(* Logix 5000 project; controller FRCFMS vendor 1 type 14 code 150 rev 33.11; software revision 33.00; part 2 of 3 *)
(* tags used below, declared in another part *)
   Additional_len : INT;
   Additional_len_read : INT;
   buff_bit_index : DINT;
   buff_byte_index : DINT;
   CMD_END : DINT;
   CMD_IN : DINT;
   CMD_LEN : DINT;
   CMD_LEN2 : INT;
   CMD_START : DINT;
   Coil_Byte_Count : DINT;
   coil_wr_index : DINT;
   Data_Received : BOOL;
   Found : BOOL;
   INT_DATA_IN : INT;
   INT_IN : INT;
   INT_STR_OUT : STRING;
   Listen_Retry_Tmr : TIMER;
   Listen_Socket_Lost : BOOL;
   Log_Old : DINT;
   Main_Read_Buffer : STR_4096[20];
   mb_bit_index : DINT;
   MB_Resp_Data : STR_462;
   MB_TMP_INT : INT;
   Modbus_Bytes : DINT;
   Modbus_CMD_Len : INT;
   Modbus_Cmd_String : STR_462;
   Modbus_ID : STRING;
   Modbus_Packet : STR_462;
   Modbus_resp_Str : STR_462;
   Modbus_Ret_CMD : STRING;
   Modbus_Ret_len : STRING;
   Modbus_Start : INT;
   Modbus_Unit : STRING;
   Next_Write : BOOL[32];
   No_Open_Sockets : BOOL;
   Nothing : BOOL;
   ONS : BOOL[64];
   RetryCreateSock : TIMER;
   RG_4x_Pos : DINT;
   RW_Instance : INT[20];
   RW_Select : DINT;
   Startup_Timer : TIMER;
   Str_Out : STR_1;
   String_Pos : INT;
   testint : DINT;
   Valid : BOOL[32];
   Valid_CMD : BOOL[32];
   Valid_Command : BOOL;
   Valid_End : BOOL;
   Valid_Len : BOOL;
   Valid_Start_Addr : BOOL;
   Valid_Value_05 : BOOL;
   W_Log_Accept : ALIAS FOR MBTU_Log_Enable.2;
   W_Log_Attribute : ALIAS FOR MBTU_Log_Enable.6;
   W_Log_Create : ALIAS FOR MBTU_Log_Enable.0;
   W_Log_Delete : ALIAS FOR MBTU_Log_Enable.5;
   W_Log_Errors : ALIAS FOR MBTU_Log_Enable.7;
   W_Log_Open : ALIAS FOR MBTU_Log_Enable.1;
   W_Log_Read : ALIAS FOR MBTU_Log_Enable.3;
   W_Log_Write : ALIAS FOR MBTU_Log_Enable.4;
   MBTI_Change_Log_MSG : MESSAGE;
   MBTI_Conn_Acc_Timeout_MSG : MESSAGE;
   MBTI_Conn_Accept_MSG : MESSAGE;
   MBTI_ConnectionsLastErrors : DINT;
   MBTI_Create_Sock_MSG : MESSAGE;
   MBTI_Delete_All_MSG : MESSAGE;
   MBTI_Instance : DINT;
   MBTI_Read_Data_MSG_00 : MESSAGE;
   MBTI_Read_Data_MSG_01 : MESSAGE;
   MBTI_Read_Data_MSG_02 : MESSAGE;
   MBTI_Read_Data_MSG_03 : MESSAGE;
   MBTI_Read_Data_MSG_04 : MESSAGE;
   MBTI_Read_Data_MSG_05 : MESSAGE;
   MBTI_Read_Data_MSG_06 : MESSAGE;
   MBTI_Read_Data_MSG_07 : MESSAGE;
   MBTI_Read_Data_MSG_08 : MESSAGE;
   MBTI_Read_Data_MSG_09 : MESSAGE;
   MBTI_Read_Done : BOOL[32];
   MBTI_Read_Resp : READ_RESP_STR[10];
   MBTI_RW_Inactivity_MSG : MESSAGE;
   MBTI_Sock_Accept_Resp : AcceptResponse;
   MBTI_Total_Open : INT;
   MBTI_Total_Open_MSG : MESSAGE;
   MBTI_Write_Data_MSG_00 : MESSAGE;
   MBTI_Write_Data_MSG_01 : MESSAGE;
   MBTI_Write_Data_MSG_02 : MESSAGE;
   MBTI_Write_Data_MSG_03 : MESSAGE;
   MBTI_Write_Data_MSG_04 : MESSAGE;
   MBTI_Write_Data_MSG_05 : MESSAGE;
   MBTI_Write_Data_MSG_06 : MESSAGE;
   MBTI_Write_Data_MSG_07 : MESSAGE;
   MBTI_Write_Data_MSG_08 : MESSAGE;
   MBTI_Write_Data_MSG_09 : MESSAGE;
   MBTI_Write_Data_Out : WRT_DATA[10];
   MBTU_Enable_MBTCP : BOOL;
   MBTU_EnetModulePort : STRING;
   MBTU_Log_Enable : DINT;
   MBTU_MB_0xx : BOOL[256];
   MBTU_MB_4xx : INT[100];
(* ModbusSlaveTCP, continued *)

ROUTINE _SUB_4x_WR   (* ladder *)
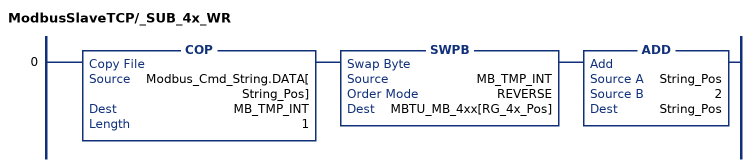
   0: COP(Modbus_Cmd_String.DATA[String_Pos],MB_TMP_INT,1)SWPB(MB_TMP_INT,REVERSE,MBTU_MB_4xx[RG_4x_Pos])ADD(String_Pos,2,String_Pos);
END_ROUTINE

ROUTINE _SUB_Byte2ST   (* ladder *)
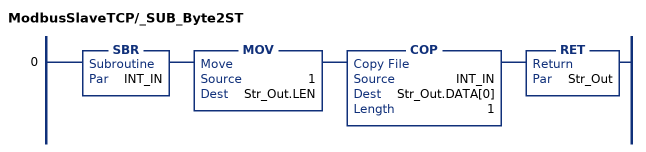
   0: SBR(INT_IN)MOV(1,Str_Out.LEN)COP(INT_IN,Str_Out.DATA[0],1)RET(Str_Out);
END_ROUTINE

ROUTINE _SUB_Int2ST   (* ladder *)
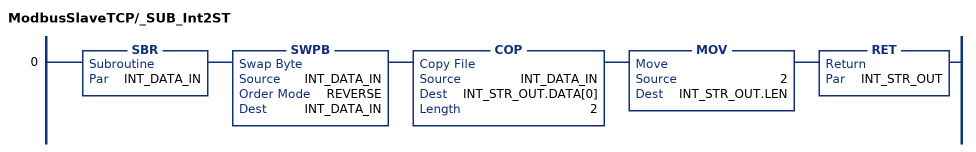
   0: SBR(INT_DATA_IN)SWPB(INT_DATA_IN,REVERSE,INT_DATA_IN)COP(INT_DATA_IN,INT_STR_OUT.DATA[0],2)MOV(2,INT_STR_OUT.LEN)RET(INT_STR_OUT);
END_ROUTINE

ROUTINE _SUB_SET_PATH   (* ladder *)
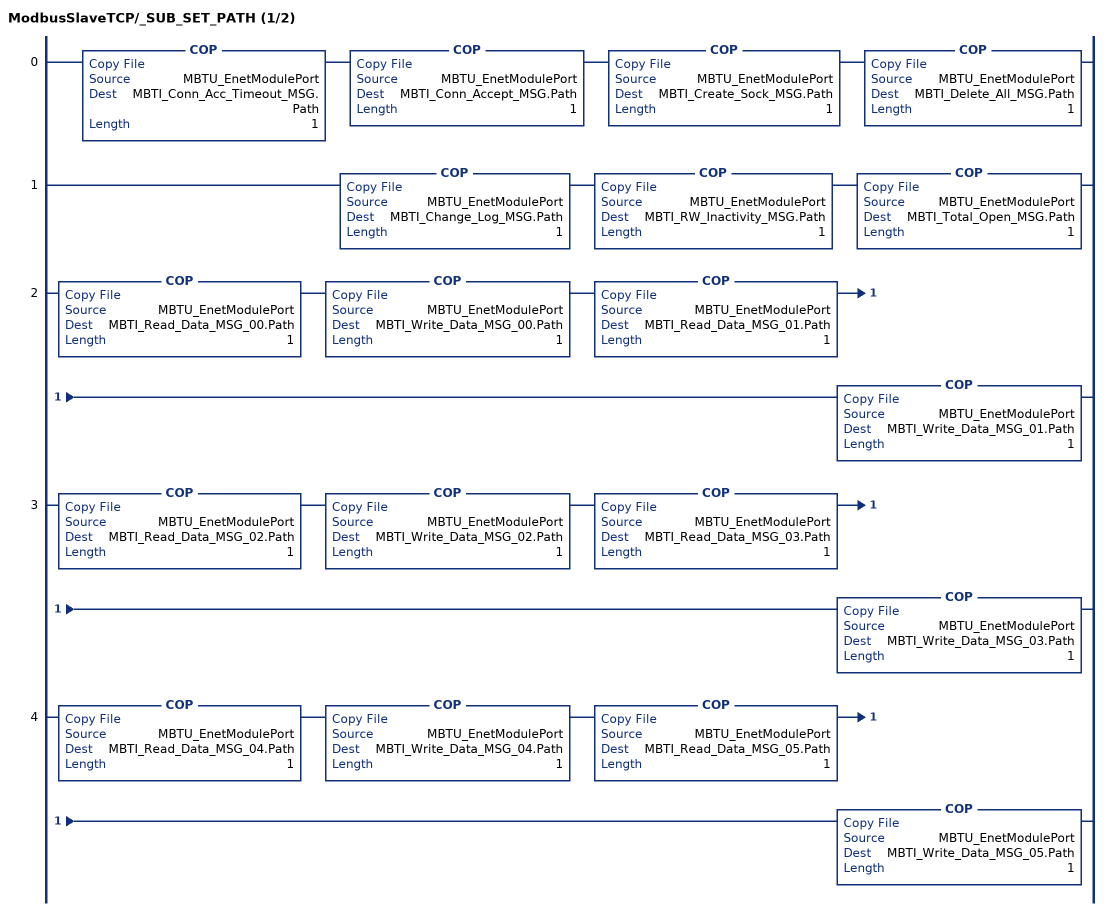
   0: COP(MBTU_EnetModulePort,MBTI_Conn_Acc_Timeout_MSG.Path,1)COP(MBTU_EnetModulePort,MBTI_Conn_Accept_MSG.Path,1)COP(MBTU_EnetModulePort,MBTI_Create_Sock_MSG.Path,1)COP(MBTU_EnetModulePort,MBTI_Delete_All_MSG.Path,1);
   1: COP(MBTU_EnetModulePort,MBTI_Change_Log_MSG.Path,1)COP(MBTU_EnetModulePort,MBTI_RW_Inactivity_MSG.Path,1)COP(MBTU_EnetModulePort,MBTI_Total_Open_MSG.Path,1);
   2: COP(MBTU_EnetModulePort,MBTI_Read_Data_MSG_00.Path,1)COP(MBTU_EnetModulePort,MBTI_Write_Data_MSG_00.Path,1)COP(MBTU_EnetModulePort,MBTI_Read_Data_MSG_01.Path,1)COP(MBTU_EnetModulePort,MBTI_Write_Data_MSG_01.Path,1);
   3: COP(MBTU_EnetModulePort,MBTI_Read_Data_MSG_02.Path,1)COP(MBTU_EnetModulePort,MBTI_Write_Data_MSG_02.Path,1)COP(MBTU_EnetModulePort,MBTI_Read_Data_MSG_03.Path,1)COP(MBTU_EnetModulePort,MBTI_Write_Data_MSG_03.Path,1);
   4: COP(MBTU_EnetModulePort,MBTI_Read_Data_MSG_04.Path,1)COP(MBTU_EnetModulePort,MBTI_Write_Data_MSG_04.Path,1)COP(MBTU_EnetModulePort,MBTI_Read_Data_MSG_05.Path,1)COP(MBTU_EnetModulePort,MBTI_Write_Data_MSG_05.Path,1);
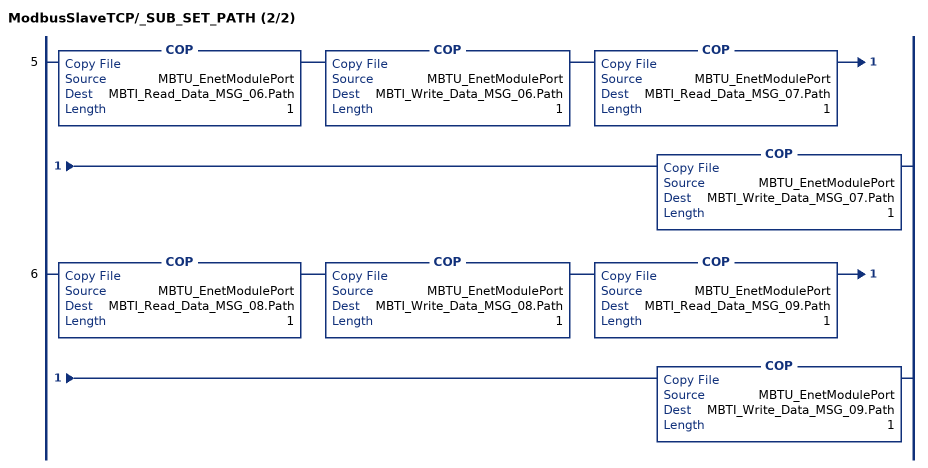
   5: COP(MBTU_EnetModulePort,MBTI_Read_Data_MSG_06.Path,1)COP(MBTU_EnetModulePort,MBTI_Write_Data_MSG_06.Path,1)COP(MBTU_EnetModulePort,MBTI_Read_Data_MSG_07.Path,1)COP(MBTU_EnetModulePort,MBTI_Write_Data_MSG_07.Path,1);
   6: COP(MBTU_EnetModulePort,MBTI_Read_Data_MSG_08.Path,1)COP(MBTU_EnetModulePort,MBTI_Write_Data_MSG_08.Path,1)COP(MBTU_EnetModulePort,MBTI_Read_Data_MSG_09.Path,1)COP(MBTU_EnetModulePort,MBTI_Write_Data_MSG_09.Path,1);
END_ROUTINE

ROUTINE Modbus_TCP_Slave   (* ladder *)
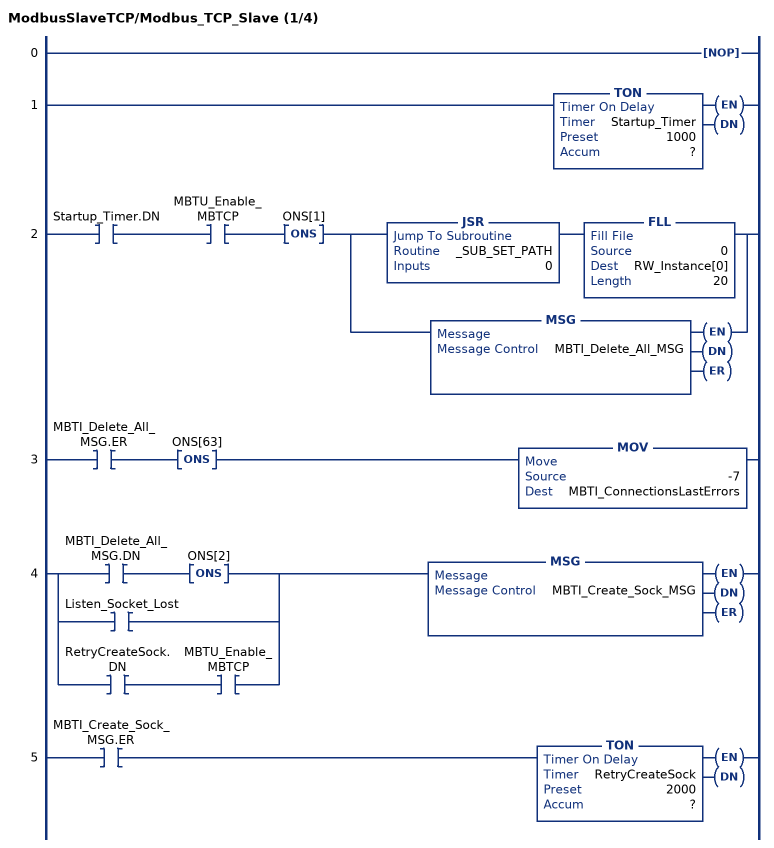
   0: NOP();
   1: TON(Startup_Timer,?,?);
   2: XIC(Startup_Timer.DN)XIC(MBTU_Enable_MBTCP)ONS(ONS[1])[JSR(_SUB_SET_PATH,0) FLL(0,RW_Instance[0],20) ,MSG(MBTI_Delete_All_MSG) ];
   3: XIC(MBTI_Delete_All_MSG.ER)ONS(ONS[63])MOV(-7,MBTI_ConnectionsLastErrors);
   4: [XIC(MBTI_Delete_All_MSG.DN) ONS(ONS[2]) ,XIC(Listen_Socket_Lost) ,XIC(RetryCreateSock.DN) XIC(MBTU_Enable_MBTCP) ]MSG(MBTI_Create_Sock_MSG);
   5: XIC(MBTI_Create_Sock_MSG.ER)TON(RetryCreateSock,?,?);
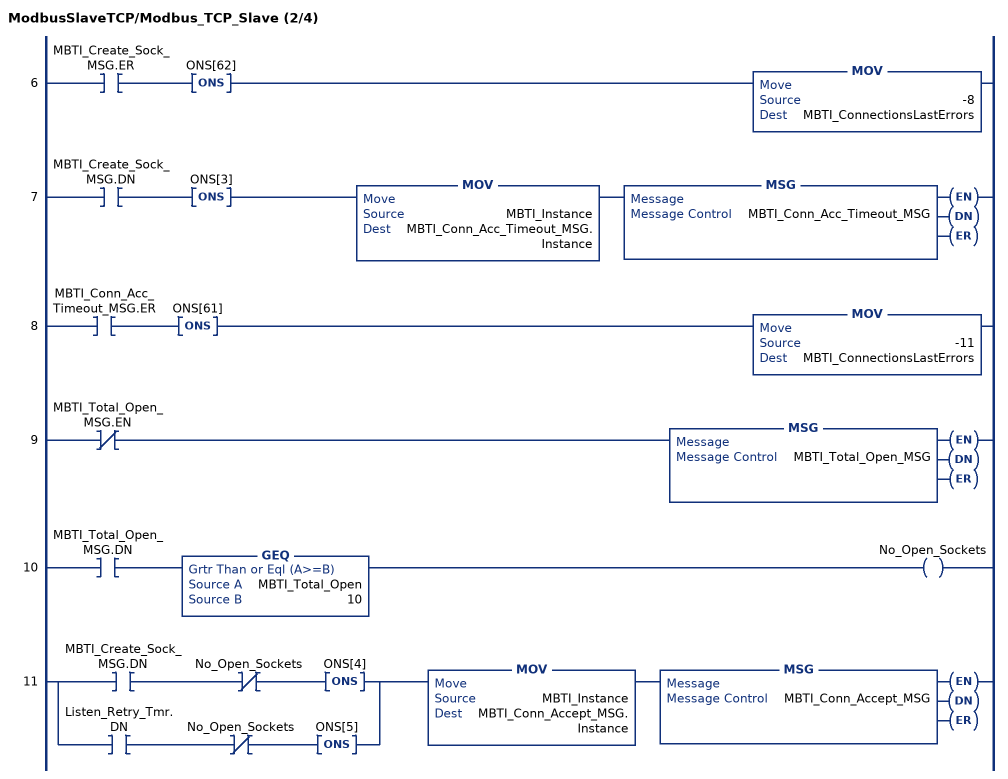
   6: XIC(MBTI_Create_Sock_MSG.ER)ONS(ONS[62])MOV(-8,MBTI_ConnectionsLastErrors);
   7: XIC(MBTI_Create_Sock_MSG.DN)ONS(ONS[3])MOV(MBTI_Instance,MBTI_Conn_Acc_Timeout_MSG.Instance)MSG(MBTI_Conn_Acc_Timeout_MSG);
   8: XIC(MBTI_Conn_Acc_Timeout_MSG.ER)ONS(ONS[61])MOV(-11,MBTI_ConnectionsLastErrors);
   9: XIO(MBTI_Total_Open_MSG.EN)MSG(MBTI_Total_Open_MSG);
   10: XIC(MBTI_Total_Open_MSG.DN)GEQ(MBTI_Total_Open,10)OTE(No_Open_Sockets);
   11: [XIC(MBTI_Create_Sock_MSG.DN) XIO(No_Open_Sockets) ONS(ONS[4]) ,XIC(Listen_Retry_Tmr.DN) XIO(No_Open_Sockets) ONS(ONS[5]) ]MOV(MBTI_Instance,MBTI_Conn_Accept_MSG.Instance)MSG(MBTI_Conn_Accept_MSG);
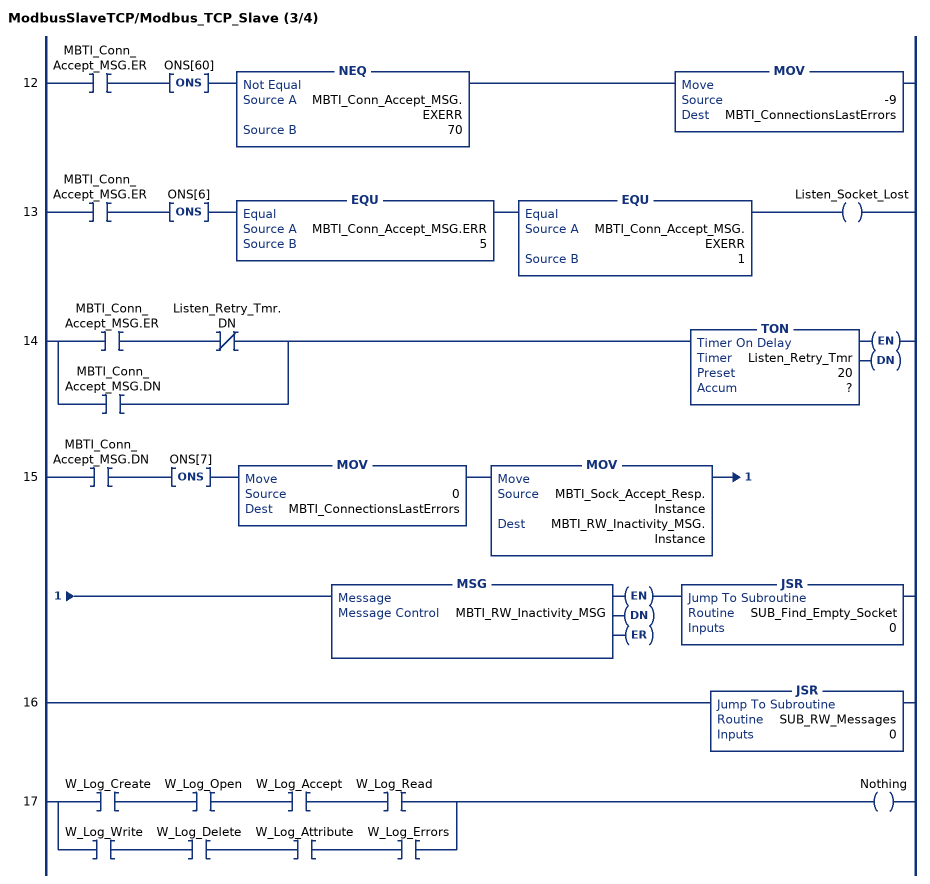
   12: XIC(MBTI_Conn_Accept_MSG.ER)ONS(ONS[60])NEQ(MBTI_Conn_Accept_MSG.EXERR,70)MOV(-9,MBTI_ConnectionsLastErrors);
   13: XIC(MBTI_Conn_Accept_MSG.ER)ONS(ONS[6])EQU(MBTI_Conn_Accept_MSG.ERR,5)EQU(MBTI_Conn_Accept_MSG.EXERR,1)OTE(Listen_Socket_Lost);
   14: [XIC(MBTI_Conn_Accept_MSG.ER) XIO(Listen_Retry_Tmr.DN) ,XIC(MBTI_Conn_Accept_MSG.DN) ]TON(Listen_Retry_Tmr,?,?);
   15: XIC(MBTI_Conn_Accept_MSG.DN)ONS(ONS[7])MOV(0,MBTI_ConnectionsLastErrors)MOV(MBTI_Sock_Accept_Resp.Instance,MBTI_RW_Inactivity_MSG.Instance)MSG(MBTI_RW_Inactivity_MSG)JSR(SUB_Find_Empty_Socket,0);
   16: JSR(SUB_RW_Messages,0);
   17: [XIC(W_Log_Create) XIC(W_Log_Open) XIC(W_Log_Accept) XIC(W_Log_Read) ,XIC(W_Log_Write) XIC(W_Log_Delete) XIC(W_Log_Attribute) XIC(W_Log_Errors) ]OTE(Nothing);
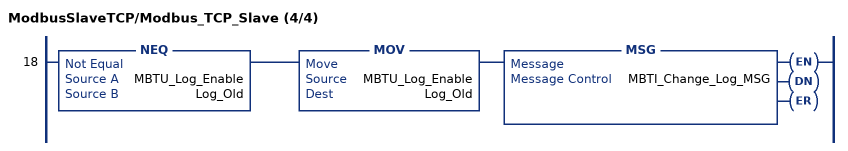
   18: NEQ(MBTU_Log_Enable,Log_Old)MOV(MBTU_Log_Enable,Log_Old)MSG(MBTI_Change_Log_MSG);
END_ROUTINE

ROUTINE Packet_Processing   (* ladder *)
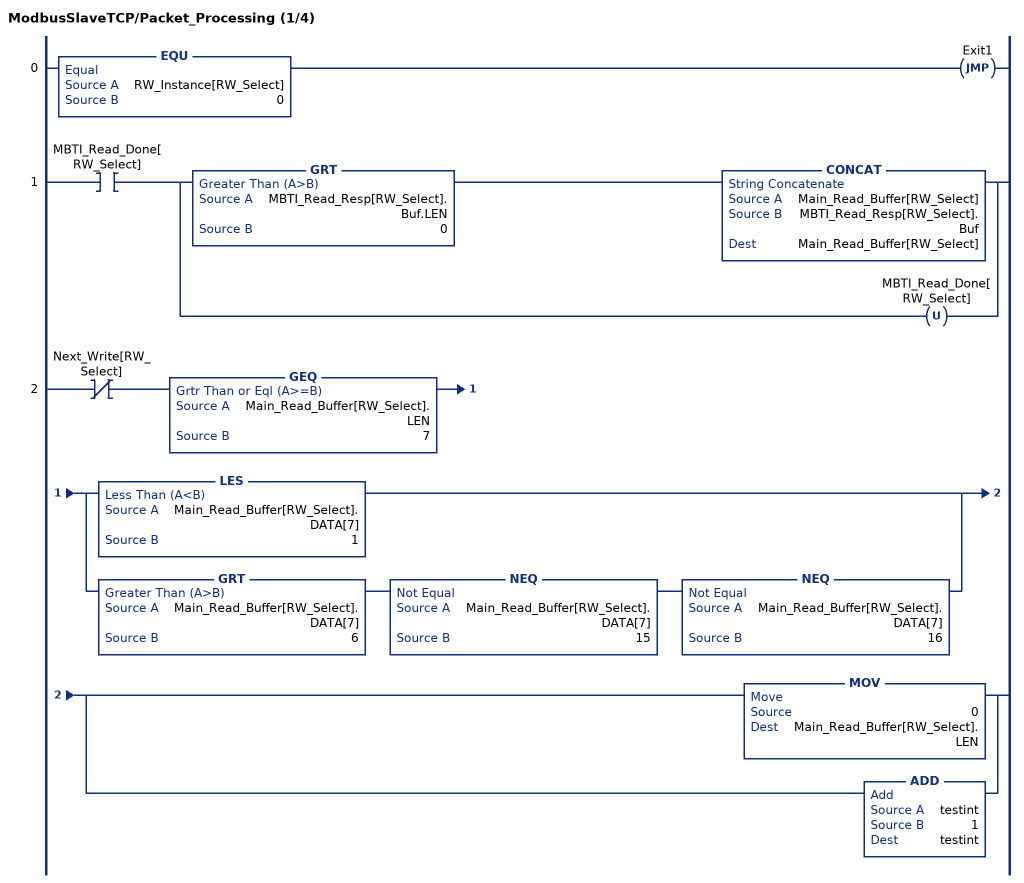
   0: EQU(RW_Instance[RW_Select],0)JMP(Exit1);
   1: XIC(MBTI_Read_Done[RW_Select])[GRT(MBTI_Read_Resp[RW_Select].Buf.LEN,0) CONCAT(Main_Read_Buffer[RW_Select],MBTI_Read_Resp[RW_Select].Buf,Main_Read_Buffer[RW_Select]) ,OTU(MBTI_Read_Done[RW_Select]) ];
   2: XIO(Next_Write[RW_Select])GEQ(Main_Read_Buffer[RW_Select].LEN,7)[LES(Main_Read_Buffer[RW_Select].DATA[7],1) ,GRT(Main_Read_Buffer[RW_Select].DATA[7],6) NEQ(Main_Read_Buffer[RW_Select].DATA[7],15) NEQ(Main_Read_Buffer[RW_Select].DATA[7],16) ][MOV(0,Main_Read_Buffer[RW_Select].LEN) ,ADD(testint,1,testint) ];
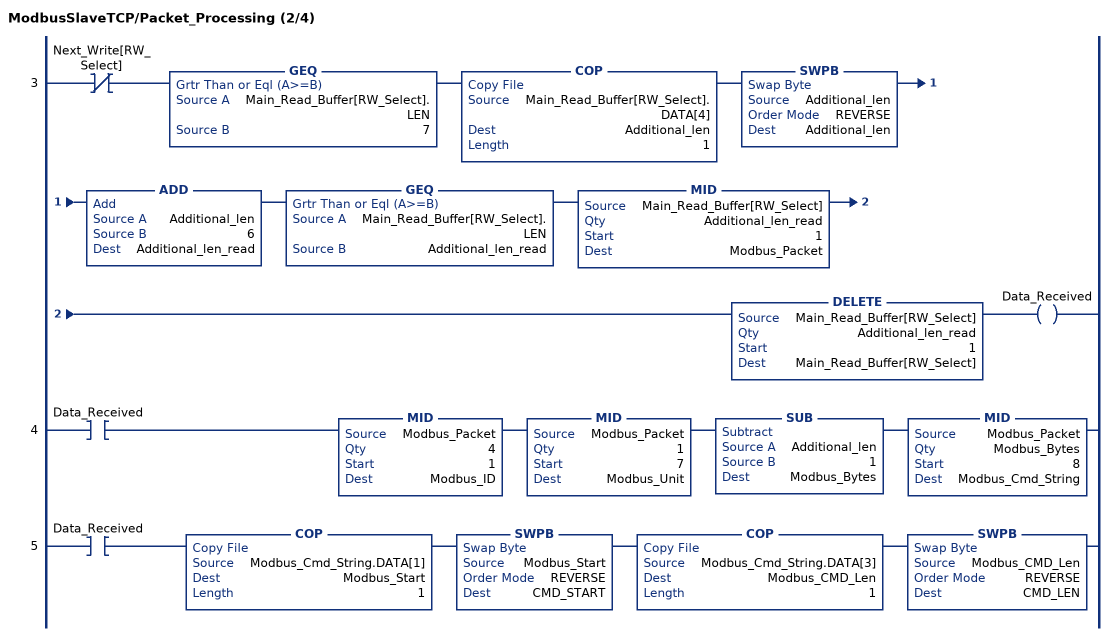
   3: XIO(Next_Write[RW_Select])GEQ(Main_Read_Buffer[RW_Select].LEN,7)COP(Main_Read_Buffer[RW_Select].DATA[4],Additional_len,1)SWPB(Additional_len,REVERSE,Additional_len)ADD(Additional_len,6,Additional_len_read)GEQ(Main_Read_Buffer[RW_Select].LEN,Additional_len_read)MID(Main_Read_Buffer[RW_Select],Additional_len_read,1,Modbus_Packet)DELETE(Main_Read_Buffer[RW_Select],Additional_len_read,1,Main_Read_Buffer[RW_Select])OTE(Data_Received);
   4: XIC(Data_Received)MID(Modbus_Packet,4,1,Modbus_ID)MID(Modbus_Packet,1,7,Modbus_Unit)SUB(Additional_len,1,Modbus_Bytes)MID(Modbus_Packet,Modbus_Bytes,8,Modbus_Cmd_String);
   5: XIC(Data_Received)COP(Modbus_Cmd_String.DATA[1],Modbus_Start,1)SWPB(Modbus_Start,REVERSE,CMD_START)COP(Modbus_Cmd_String.DATA[3],Modbus_CMD_Len,1)SWPB(Modbus_CMD_Len,REVERSE,CMD_LEN);
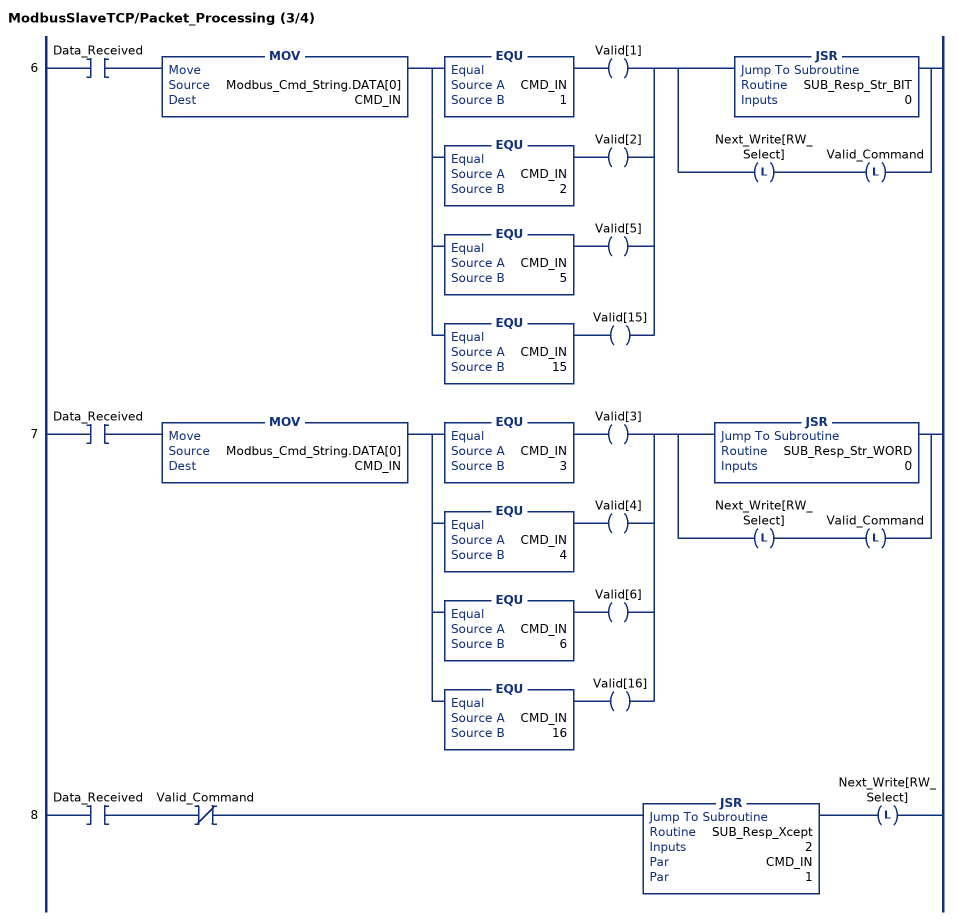
   6: XIC(Data_Received)MOV(Modbus_Cmd_String.DATA[0],CMD_IN)[EQU(CMD_IN,1) OTE(Valid[1]) ,EQU(CMD_IN,2) OTE(Valid[2]) ,EQU(CMD_IN,5) OTE(Valid[5]) ,EQU(CMD_IN,15) OTE(Valid[15]) ][JSR(SUB_Resp_Str_BIT,0) ,OTL(Next_Write[RW_Select]) OTL(Valid_Command) ];
   7: XIC(Data_Received)MOV(Modbus_Cmd_String.DATA[0],CMD_IN)[EQU(CMD_IN,3) OTE(Valid[3]) ,EQU(CMD_IN,4) OTE(Valid[4]) ,EQU(CMD_IN,6) OTE(Valid[6]) ,EQU(CMD_IN,16) OTE(Valid[16]) ][JSR(SUB_Resp_Str_WORD,0) ,OTL(Next_Write[RW_Select]) OTL(Valid_Command) ];
   8: XIC(Data_Received)XIO(Valid_Command)JSR(SUB_Resp_Xcept,2,CMD_IN,1)OTL(Next_Write[RW_Select]);
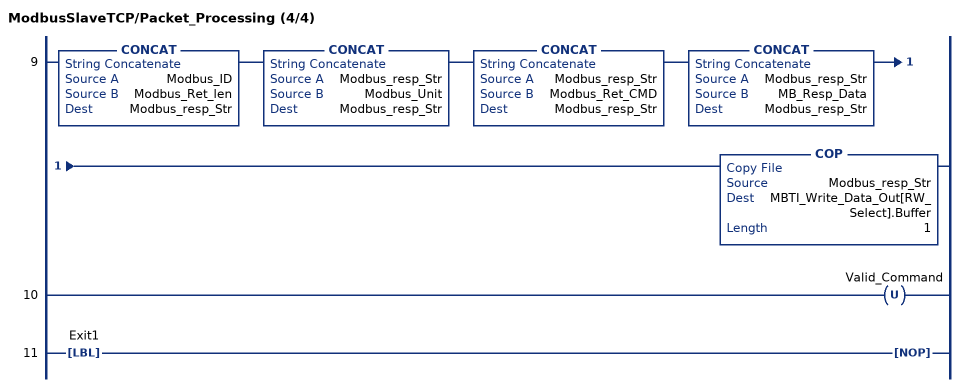
   9: CONCAT(Modbus_ID,Modbus_Ret_len,Modbus_resp_Str)CONCAT(Modbus_resp_Str,Modbus_Unit,Modbus_resp_Str)CONCAT(Modbus_resp_Str,Modbus_Ret_CMD,Modbus_resp_Str)CONCAT(Modbus_resp_Str,MB_Resp_Data,Modbus_resp_Str)COP(Modbus_resp_Str,MBTI_Write_Data_Out[RW_Select].Buffer,1);
   10: OTU(Valid_Command);
   11: LBL(Exit1)NOP();
END_ROUTINE

ROUTINE SUB_Find_Empty_Socket   (* ladder *)
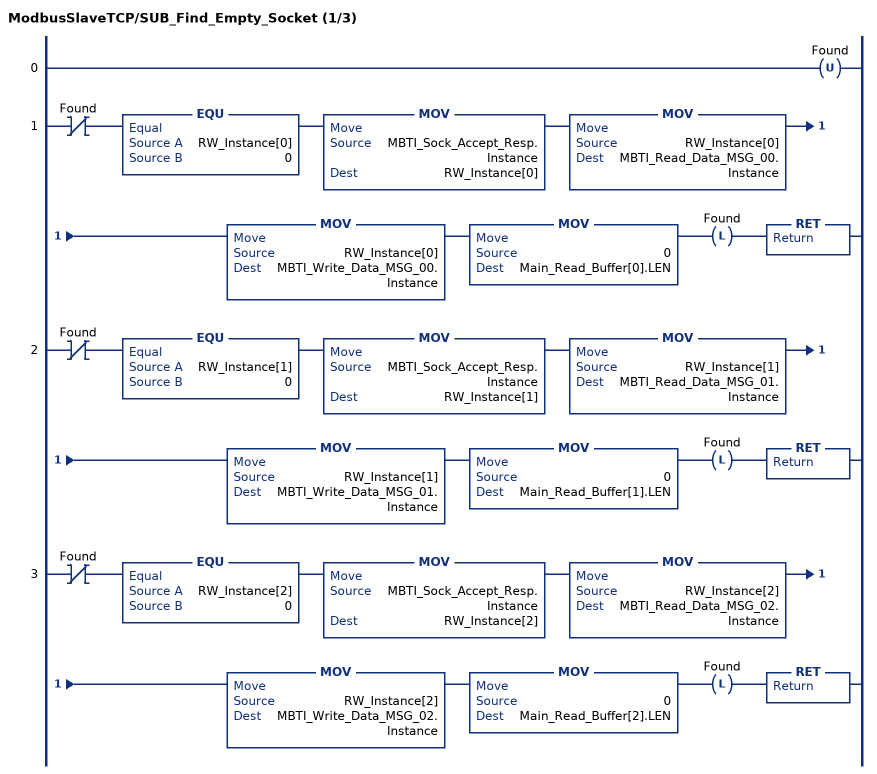
   0: OTU(Found);
   1: XIO(Found)EQU(RW_Instance[0],0)MOV(MBTI_Sock_Accept_Resp.Instance,RW_Instance[0])MOV(RW_Instance[0],MBTI_Read_Data_MSG_00.Instance)MOV(RW_Instance[0],MBTI_Write_Data_MSG_00.Instance)MOV(0,Main_Read_Buffer[0].LEN)OTL(Found)RET();
   2: XIO(Found)EQU(RW_Instance[1],0)MOV(MBTI_Sock_Accept_Resp.Instance,RW_Instance[1])MOV(RW_Instance[1],MBTI_Read_Data_MSG_01.Instance)MOV(RW_Instance[1],MBTI_Write_Data_MSG_01.Instance)MOV(0,Main_Read_Buffer[1].LEN)OTL(Found)RET();
   3: XIO(Found)EQU(RW_Instance[2],0)MOV(MBTI_Sock_Accept_Resp.Instance,RW_Instance[2])MOV(RW_Instance[2],MBTI_Read_Data_MSG_02.Instance)MOV(RW_Instance[2],MBTI_Write_Data_MSG_02.Instance)MOV(0,Main_Read_Buffer[2].LEN)OTL(Found)RET();
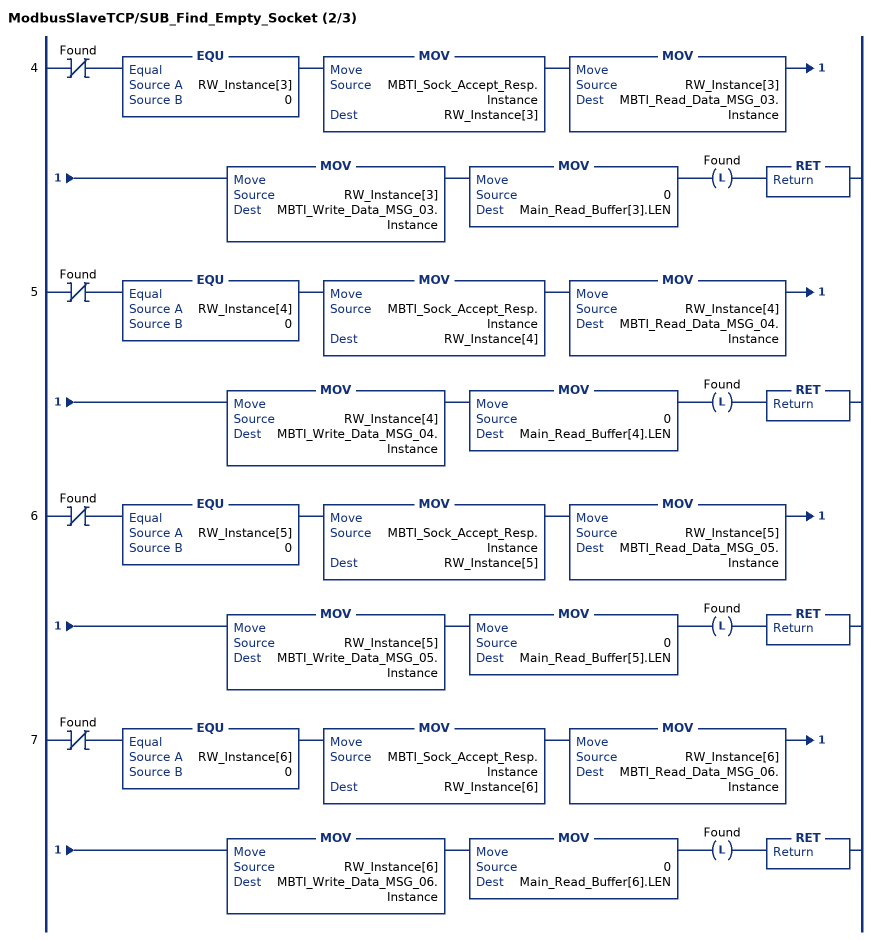
   4: XIO(Found)EQU(RW_Instance[3],0)MOV(MBTI_Sock_Accept_Resp.Instance,RW_Instance[3])MOV(RW_Instance[3],MBTI_Read_Data_MSG_03.Instance)MOV(RW_Instance[3],MBTI_Write_Data_MSG_03.Instance)MOV(0,Main_Read_Buffer[3].LEN)OTL(Found)RET();
   5: XIO(Found)EQU(RW_Instance[4],0)MOV(MBTI_Sock_Accept_Resp.Instance,RW_Instance[4])MOV(RW_Instance[4],MBTI_Read_Data_MSG_04.Instance)MOV(RW_Instance[4],MBTI_Write_Data_MSG_04.Instance)MOV(0,Main_Read_Buffer[4].LEN)OTL(Found)RET();
   6: XIO(Found)EQU(RW_Instance[5],0)MOV(MBTI_Sock_Accept_Resp.Instance,RW_Instance[5])MOV(RW_Instance[5],MBTI_Read_Data_MSG_05.Instance)MOV(RW_Instance[5],MBTI_Write_Data_MSG_05.Instance)MOV(0,Main_Read_Buffer[5].LEN)OTL(Found)RET();
   7: XIO(Found)EQU(RW_Instance[6],0)MOV(MBTI_Sock_Accept_Resp.Instance,RW_Instance[6])MOV(RW_Instance[6],MBTI_Read_Data_MSG_06.Instance)MOV(RW_Instance[6],MBTI_Write_Data_MSG_06.Instance)MOV(0,Main_Read_Buffer[6].LEN)OTL(Found)RET();
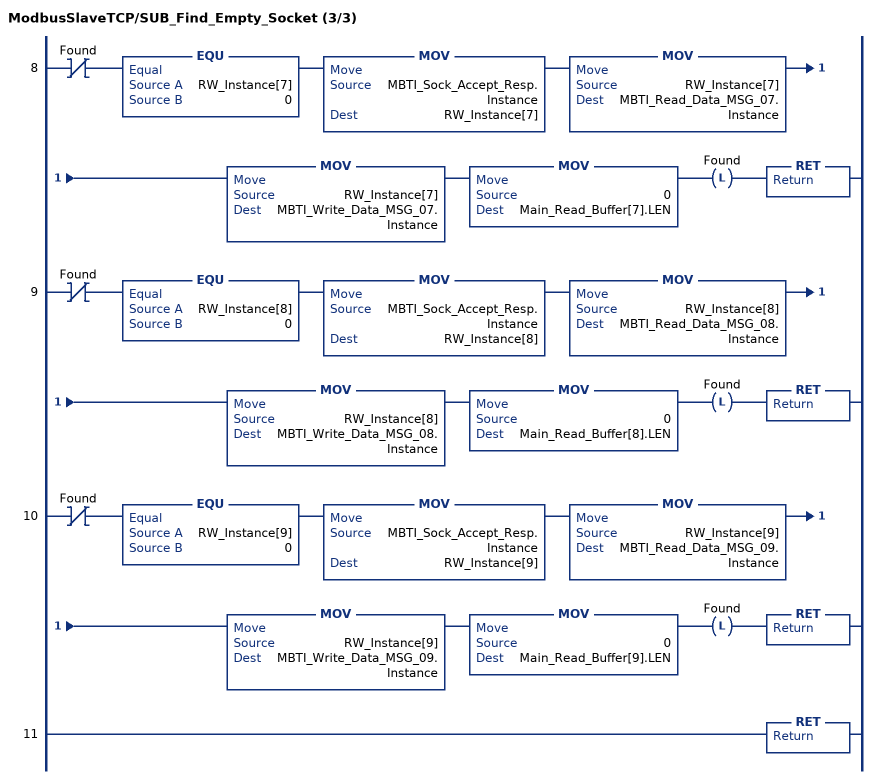
   8: XIO(Found)EQU(RW_Instance[7],0)MOV(MBTI_Sock_Accept_Resp.Instance,RW_Instance[7])MOV(RW_Instance[7],MBTI_Read_Data_MSG_07.Instance)MOV(RW_Instance[7],MBTI_Write_Data_MSG_07.Instance)MOV(0,Main_Read_Buffer[7].LEN)OTL(Found)RET();
   9: XIO(Found)EQU(RW_Instance[8],0)MOV(MBTI_Sock_Accept_Resp.Instance,RW_Instance[8])MOV(RW_Instance[8],MBTI_Read_Data_MSG_08.Instance)MOV(RW_Instance[8],MBTI_Write_Data_MSG_08.Instance)MOV(0,Main_Read_Buffer[8].LEN)OTL(Found)RET();
   10: XIO(Found)EQU(RW_Instance[9],0)MOV(MBTI_Sock_Accept_Resp.Instance,RW_Instance[9])MOV(RW_Instance[9],MBTI_Read_Data_MSG_09.Instance)MOV(RW_Instance[9],MBTI_Write_Data_MSG_09.Instance)MOV(0,Main_Read_Buffer[9].LEN)OTL(Found)RET();
   11: RET();
END_ROUTINE

ROUTINE SUB_Resp_Str_BIT   (* ladder *)
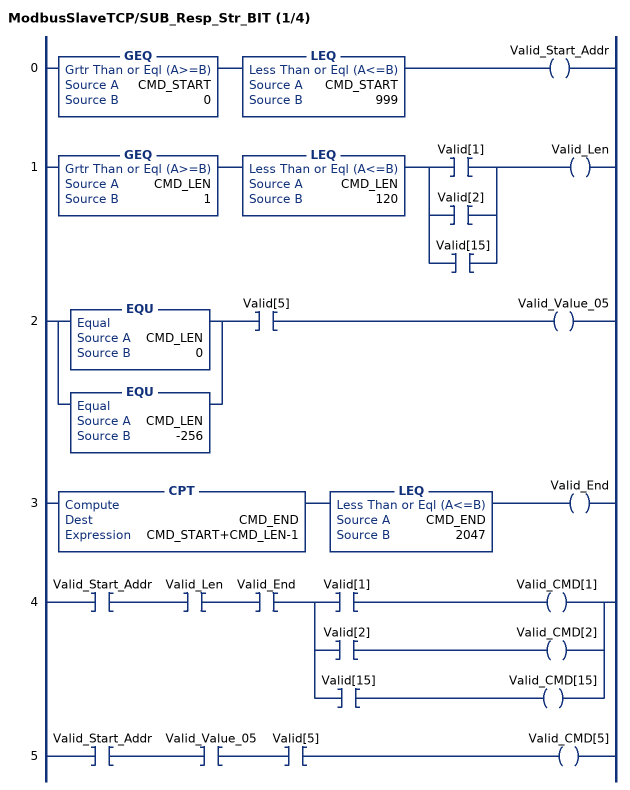
   0: GEQ(CMD_START,0)LEQ(CMD_START,999)OTE(Valid_Start_Addr);
   1: GEQ(CMD_LEN,1)LEQ(CMD_LEN,120)[XIC(Valid[1]) ,XIC(Valid[2]) ,XIC(Valid[15]) ]OTE(Valid_Len);
   2: [EQU(CMD_LEN,0) ,EQU(CMD_LEN,-256) ]XIC(Valid[5])OTE(Valid_Value_05);
   3: CPT(CMD_END,CMD_START+CMD_LEN-1)LEQ(CMD_END,2047)OTE(Valid_End);
   4: XIC(Valid_Start_Addr)XIC(Valid_Len)XIC(Valid_End)[XIC(Valid[1]) OTE(Valid_CMD[1]) ,XIC(Valid[2]) OTE(Valid_CMD[2]) ,XIC(Valid[15]) OTE(Valid_CMD[15]) ];
   5: XIC(Valid_Start_Addr)XIC(Valid_Value_05)XIC(Valid[5])OTE(Valid_CMD[5]);
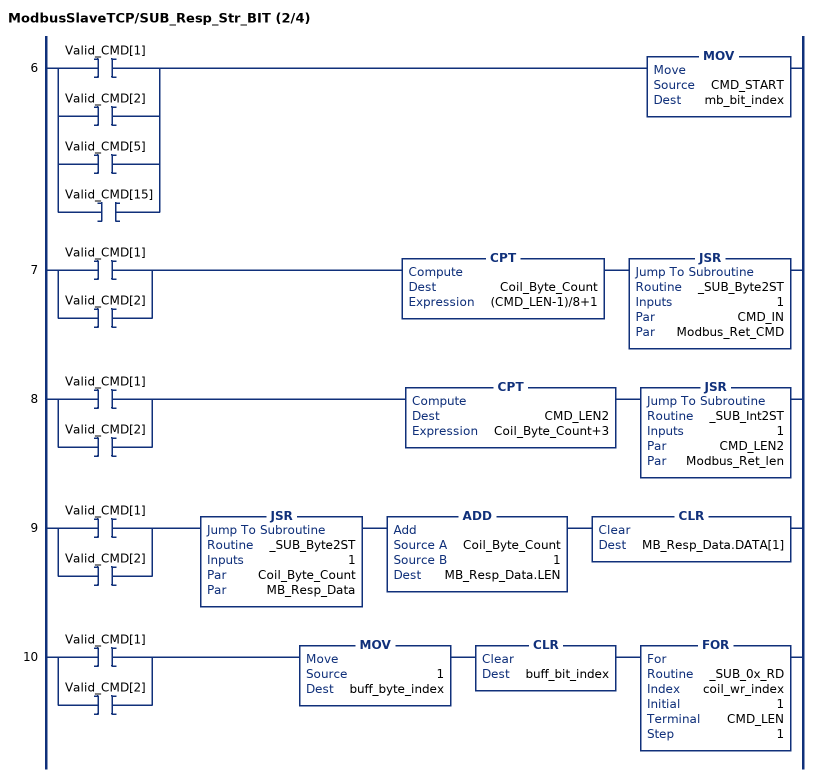
   6: [XIC(Valid_CMD[1]) ,XIC(Valid_CMD[2]) ,XIC(Valid_CMD[5]) ,XIC(Valid_CMD[15]) ]MOV(CMD_START,mb_bit_index);
   7: [XIC(Valid_CMD[1]) ,XIC(Valid_CMD[2]) ]CPT(Coil_Byte_Count,(CMD_LEN-1)/8+1)JSR(_SUB_Byte2ST,1,CMD_IN,Modbus_Ret_CMD);
   8: [XIC(Valid_CMD[1]) ,XIC(Valid_CMD[2]) ]CPT(CMD_LEN2,Coil_Byte_Count+3)JSR(_SUB_Int2ST,1,CMD_LEN2,Modbus_Ret_len);
   9: [XIC(Valid_CMD[1]) ,XIC(Valid_CMD[2]) ]JSR(_SUB_Byte2ST,1,Coil_Byte_Count,MB_Resp_Data)ADD(Coil_Byte_Count,1,MB_Resp_Data.LEN)CLR(MB_Resp_Data.DATA[1]);
   10: [XIC(Valid_CMD[1]) ,XIC(Valid_CMD[2]) ]MOV(1,buff_byte_index)CLR(buff_bit_index)FOR(_SUB_0x_RD,coil_wr_index,1,CMD_LEN,1);
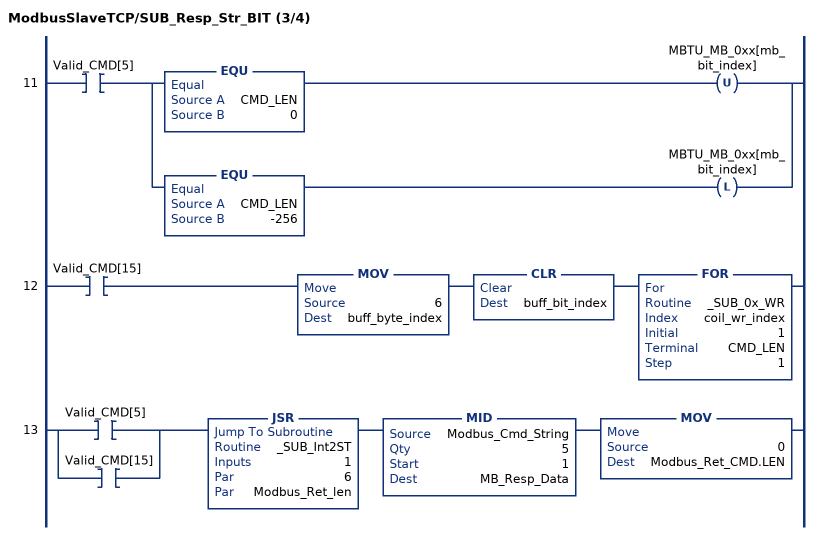
   11: XIC(Valid_CMD[5])[EQU(CMD_LEN,0) OTU(MBTU_MB_0xx[mb_bit_index]) ,EQU(CMD_LEN,-256) OTL(MBTU_MB_0xx[mb_bit_index]) ];
   12: XIC(Valid_CMD[15])MOV(6,buff_byte_index)CLR(buff_bit_index)FOR(_SUB_0x_WR,coil_wr_index,1,CMD_LEN,1);
   13: [XIC(Valid_CMD[5]) ,XIC(Valid_CMD[15]) ]JSR(_SUB_Int2ST,1,6,Modbus_Ret_len)MID(Modbus_Cmd_String,5,1,MB_Resp_Data)MOV(0,Modbus_Ret_CMD.LEN);
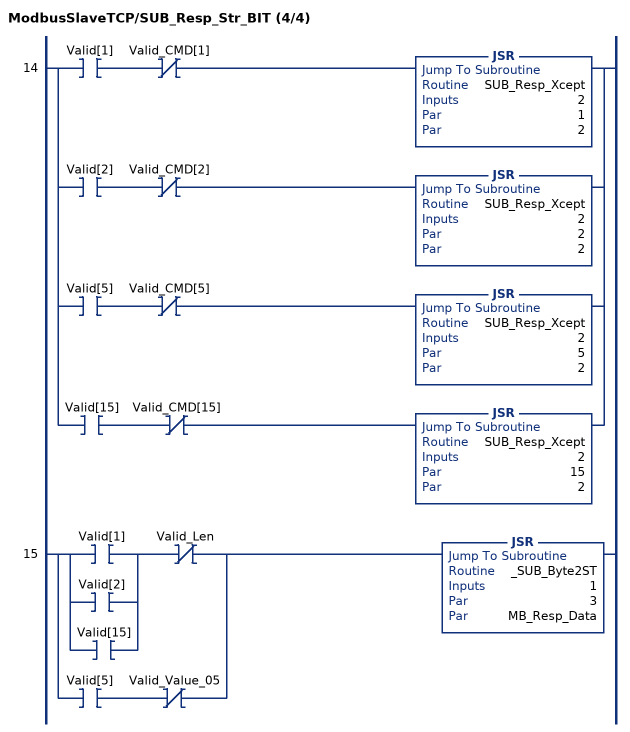
   14: [XIC(Valid[1]) XIO(Valid_CMD[1]) JSR(SUB_Resp_Xcept,2,1,2) ,XIC(Valid[2]) XIO(Valid_CMD[2]) JSR(SUB_Resp_Xcept,2,2,2) ,XIC(Valid[5]) XIO(Valid_CMD[5]) JSR(SUB_Resp_Xcept,2,5,2) ,XIC(Valid[15]) XIO(Valid_CMD[15]) JSR(SUB_Resp_Xcept,2,15,2) ];
   15: [[XIC(Valid[1]) ,XIC(Valid[2]) ,XIC(Valid[15]) ] XIO(Valid_Len) ,XIC(Valid[5]) XIO(Valid_Value_05) ]JSR(_SUB_Byte2ST,1,3,MB_Resp_Data);
END_ROUTINE
